(* CODESYS project Error_Message_Enum.export

Project tree, tasks and I/O mapping:
  Error_Message_Enum/
    data type Error_Message
*)

// Error_Message_Enum/Error_Message
{attribute 'qualified_only'}
{attribute 'strict'}
TYPE Error_Message :
(
	Err_None := 0,
	
	Err_AuxAxis_Movement_Cannot_read_virture_robot_position := 10,	// gesture block not reading robot position
	Err_Gesture_Type_Hand_Pos_Not_Given := 20,	// gesture block not given position
	Err_AuxAxis_Movement_Block_err := 30,	// gesture block first reset movement block err
	Err_Gesture_Type_Cycle_mov_block_err := 40,	// gesture block cycle movement block err
	
	Err_PowerOn_Block_Err := 50,
	Err_PowerOn_TimeOut := 51,
	
	Err_Power_Reset_Block_Err := 60,
	Err_Power_Reset_TimeOut := 61,
	
	Err_Group_Enable_Block_Err := 70,
	Err_Group_Enable_TimeOut := 71
);
END_TYPE
